{attribute 'qualified_only'}
VAR_GLOBAL CONSTANT
	MAX_SQL_LENGTH : UDINT := 10000;
END_VAR

(* stored: Version 1.1.0.1, ProductVersion 3.1.4020.3
   GVL GVL_DATABASE_LIB: Id {1987a635-9145-4d42-9345-9631ac25c7de} *)
